SUBAPPLICATION ManyOutputsSIFB100 (* Subapplication Type *)
  (* Standard: 61499-2 *)
  (* Version 1.0, 2025-05-03, cochicde *)
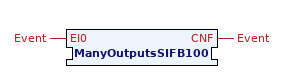
  EVENT_INPUT
    EI0;
  END_EVENT
  EVENT_OUTPUT
    CNF;
  END_EVENT
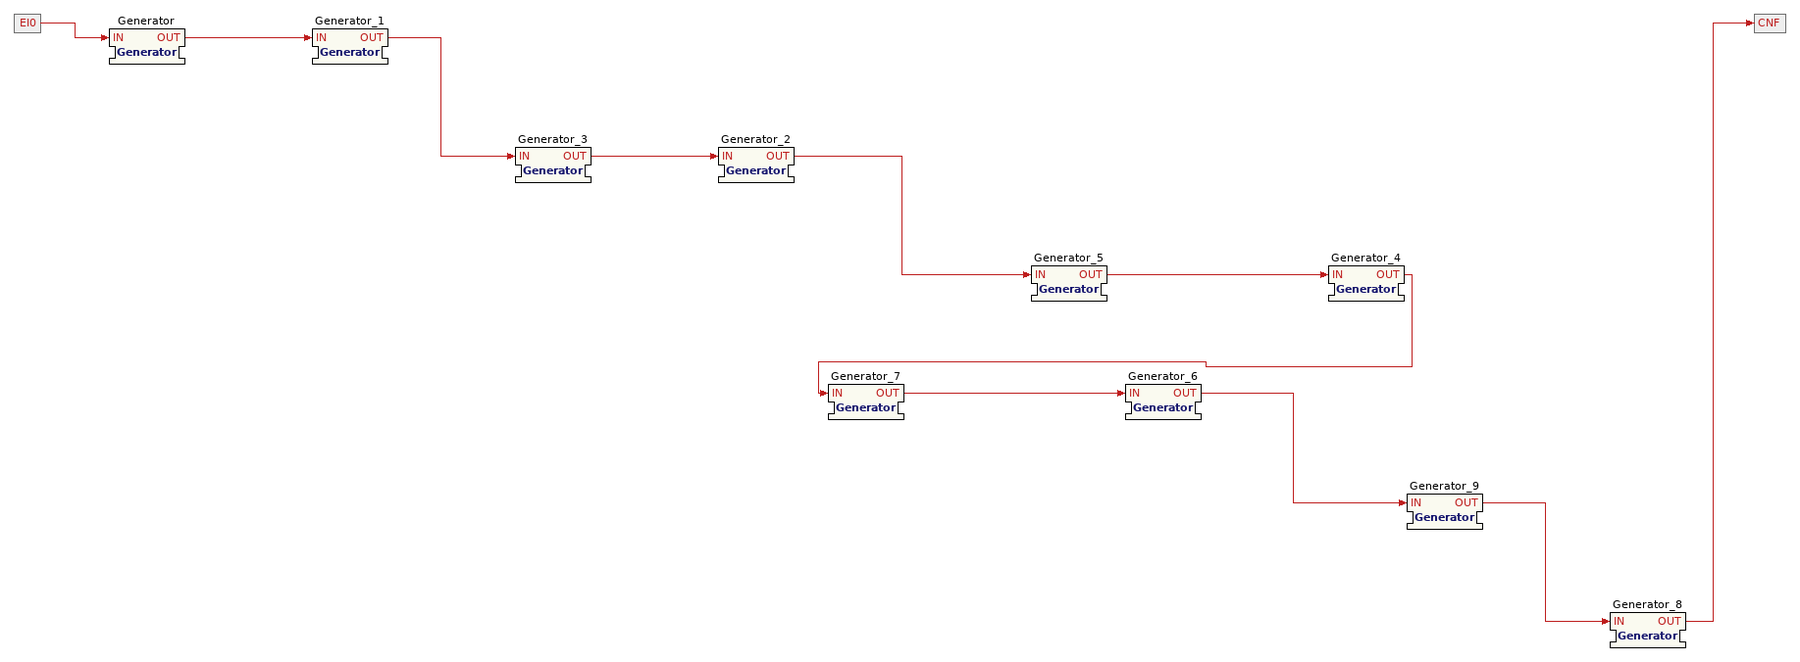
  FBS
    Generator_7 : performance::Generator;
    Generator_3 : performance::Generator;
    Generator_1 : performance::Generator;
    Generator_5 : performance::Generator;
    Generator_8 : performance::Generator;
    Generator_9 : performance::Generator;
    Generator_2 : performance::Generator;
    Generator : performance::Generator;
    Generator_6 : performance::Generator;
    Generator_4 : performance::Generator;
  END_FBS
  EVENT_CONNECTIONS
    Generator_4.OUT TO Generator_7.IN;
    Generator_7.OUT TO Generator_6.IN;
    Generator_1.OUT TO Generator_3.IN;
    Generator_3.OUT TO Generator_2.IN;
    Generator.OUT TO Generator_1.IN;
    Generator_2.OUT TO Generator_5.IN;
    Generator_5.OUT TO Generator_4.IN;
    Generator_9.OUT TO Generator_8.IN;
    Generator_6.OUT TO Generator_9.IN;
    Generator_8.OUT TO CNF;
    EI0 TO Generator.IN;
  END_CONNECTIONS
END_SUBAPPLICATION
